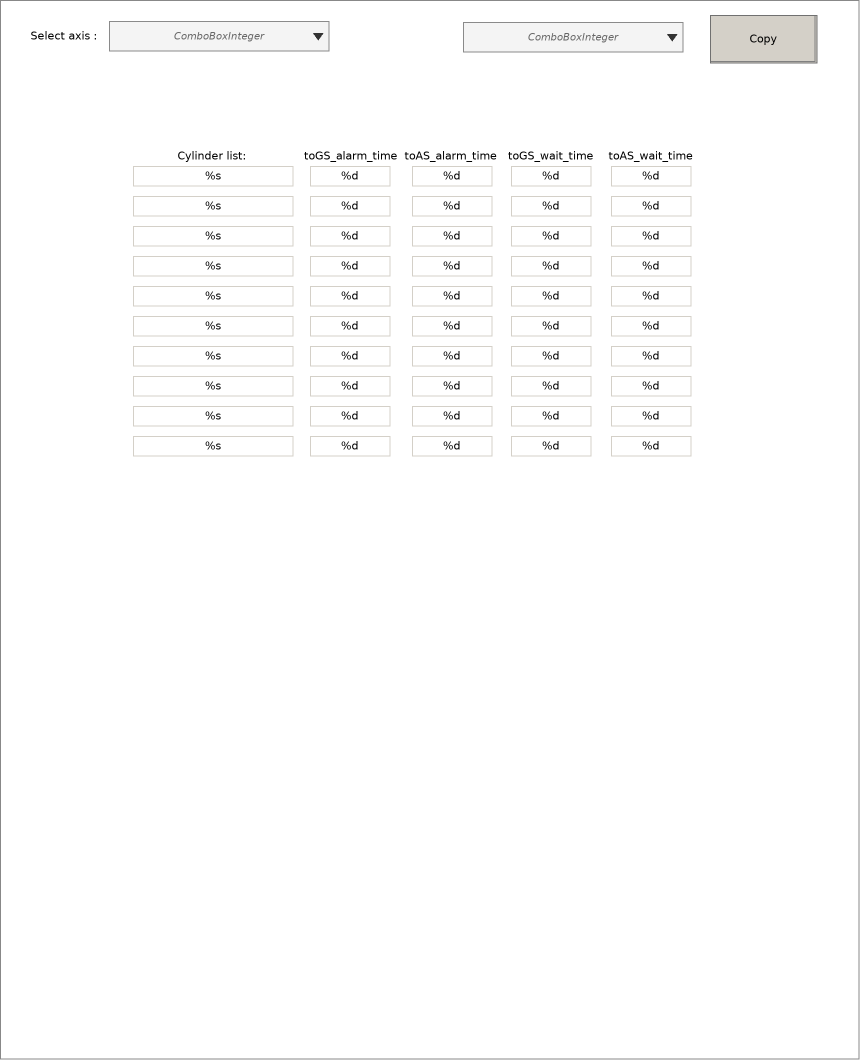
VISUALIZATION VISU_Cylinder2PosConfig  // 860x1060
    Label (165,146 94x20), "Cylinder list:"
    Label (22,21 84x30), "Select axis :"
    Label (401,146 100x20), "toAS_alarm_time"
    Label (501,146 100x20), "toGS_wait_time"
    Label (601,146 100x20), "toAS_wait_time"
    ComboBoxInteger (109,21 220x30), variable: HMI.iSelectCylinder
    Label (301,146 100x20), "toGS_alarm_time"
    Textfield (133,166 160x20), "%s", text variable: HMI.cylinderNames[HMI.iSelectCylinder][0]
    Textfield (133,196 160x20), "%s", text variable: HMI.cylinderNames[HMI.iSelectCylinder][1]
    Textfield (133,226 160x20), "%s", text variable: HMI.cylinderNames[HMI.iSelectCylinder][2]
    Textfield (133,256 160x20), "%s", text variable: HMI.cylinderNames[HMI.iSelectCylinder][3]
    Textfield (133,286 160x20), "%s", text variable: HMI.cylinderNames[HMI.iSelectCylinder][4]
    Textfield (133,316 160x20), "%s", text variable: HMI.cylinderNames[HMI.iSelectCylinder][5]
    Textfield (133,346 160x20), "%s", text variable: HMI.cylinderNames[HMI.iSelectCylinder][6]
    Textfield (133,376 160x20), "%s", text variable: HMI.cylinderNames[HMI.iSelectCylinder][7]
    Textfield (133,406 160x20), "%s", text variable: HMI.cylinderNames[HMI.iSelectCylinder][8]
    Textfield (133,436 160x20), "%s", text variable: HMI.cylinderNames[HMI.iSelectCylinder][9]
    ComboBoxInteger (463,22 220x30), variable: HMI.iSelectCylinderCopy
    Button (710,15 107x48), "Copy"
        tap HMI.btCopyCylinderCfg.button
    Textfield (310,166 80x20), "%d", text variable: _20_AUTO.recipe.cylinder2Pos[HMI.iSelectCylinder][0].toGS_alarm_time
        OnMouseDown: write the text variable via Default
    Textfield (412,166 80x20), "%d", text variable: _20_AUTO.recipe.cylinder2Pos[HMI.iSelectCylinder][0].toAS_alarm_time
        OnMouseDown: write the text variable via Default
    Textfield (511,166 80x20), "%d", text variable: _20_AUTO.recipe.cylinder2Pos[HMI.iSelectCylinder][0].toGS_wait_time
        OnMouseDown: write the text variable via Default
    Textfield (611,166 80x20), "%d", text variable: _20_AUTO.recipe.cylinder2Pos[HMI.iSelectCylinder][0].toAS_wait_time
        OnMouseDown: write the text variable via Default
    Textfield (310,196 80x20), "%d", text variable: _20_AUTO.recipe.cylinder2Pos[HMI.iSelectCylinder][1].toGS_alarm_time
        OnMouseDown: write the text variable via Default
    Textfield (412,196 80x20), "%d", text variable: _20_AUTO.recipe.cylinder2Pos[HMI.iSelectCylinder][1].toAS_alarm_time
        OnMouseDown: write the text variable via Default
    Textfield (511,196 80x20), "%d", text variable: _20_AUTO.recipe.cylinder2Pos[HMI.iSelectCylinder][1].toGS_wait_time
        OnMouseDown: write the text variable via Default
    Textfield (611,196 80x20), "%d", text variable: _20_AUTO.recipe.cylinder2Pos[HMI.iSelectCylinder][1].toAS_wait_time
        OnMouseDown: write the text variable via Default
    Textfield (310,226 80x20), "%d", text variable: _20_AUTO.recipe.cylinder2Pos[HMI.iSelectCylinder][2].toGS_alarm_time
        OnMouseDown: write the text variable via Default
    Textfield (412,226 80x20), "%d", text variable: _20_AUTO.recipe.cylinder2Pos[HMI.iSelectCylinder][2].toAS_alarm_time
        OnMouseDown: write the text variable via Default
    Textfield (511,226 80x20), "%d", text variable: _20_AUTO.recipe.cylinder2Pos[HMI.iSelectCylinder][2].toGS_wait_time
        OnMouseDown: write the text variable via Default
    Textfield (611,226 80x20), "%d", text variable: _20_AUTO.recipe.cylinder2Pos[HMI.iSelectCylinder][2].toAS_wait_time
        OnMouseDown: write the text variable via Default
    Textfield (310,256 80x20), "%d", text variable: _20_AUTO.recipe.cylinder2Pos[HMI.iSelectCylinder][3].toGS_alarm_time
        OnMouseDown: write the text variable via Default
    Textfield (412,256 80x20), "%d", text variable: _20_AUTO.recipe.cylinder2Pos[HMI.iSelectCylinder][3].toAS_alarm_time
        OnMouseDown: write the text variable via Default
    Textfield (511,256 80x20), "%d", text variable: _20_AUTO.recipe.cylinder2Pos[HMI.iSelectCylinder][3].toGS_wait_time
        OnMouseDown: write the text variable via Default
    Textfield (611,256 80x20), "%d", text variable: _20_AUTO.recipe.cylinder2Pos[HMI.iSelectCylinder][3].toAS_wait_time
        OnMouseDown: write the text variable via Default
    Textfield (310,286 80x20), "%d", text variable: _20_AUTO.recipe.cylinder2Pos[HMI.iSelectCylinder][4].toGS_alarm_time
        OnMouseDown: write the text variable via Default
    Textfield (412,286 80x20), "%d", text variable: _20_AUTO.recipe.cylinder2Pos[HMI.iSelectCylinder][4].toAS_alarm_time
        OnMouseDown: write the text variable via Default
    Textfield (511,286 80x20), "%d", text variable: _20_AUTO.recipe.cylinder2Pos[HMI.iSelectCylinder][4].toGS_wait_time
        OnMouseDown: write the text variable via Default
    Textfield (611,286 80x20), "%d", text variable: _20_AUTO.recipe.cylinder2Pos[HMI.iSelectCylinder][4].toAS_wait_time
        OnMouseDown: write the text variable via Default
    Textfield (310,316 80x20), "%d", text variable: _20_AUTO.recipe.cylinder2Pos[HMI.iSelectCylinder][5].toGS_alarm_time
        OnMouseDown: write the text variable via Default
    Textfield (412,316 80x20), "%d", text variable: _20_AUTO.recipe.cylinder2Pos[HMI.iSelectCylinder][5].toAS_alarm_time
        OnMouseDown: write the text variable via Default
    Textfield (511,316 80x20), "%d", text variable: _20_AUTO.recipe.cylinder2Pos[HMI.iSelectCylinder][5].toGS_wait_time
        OnMouseDown: write the text variable via Default
    Textfield (611,316 80x20), "%d", text variable: _20_AUTO.recipe.cylinder2Pos[HMI.iSelectCylinder][5].toAS_wait_time
        OnMouseDown: write the text variable via Default
    Textfield (310,346 80x20), "%d", text variable: _20_AUTO.recipe.cylinder2Pos[HMI.iSelectCylinder][6].toGS_alarm_time
        OnMouseDown: write the text variable via Default
    Textfield (412,346 80x20), "%d", text variable: _20_AUTO.recipe.cylinder2Pos[HMI.iSelectCylinder][6].toAS_alarm_time
        OnMouseDown: write the text variable via Default
    Textfield (511,346 80x20), "%d", text variable: _20_AUTO.recipe.cylinder2Pos[HMI.iSelectCylinder][6].toGS_wait_time
        OnMouseDown: write the text variable via Default
    Textfield (611,346 80x20), "%d", text variable: _20_AUTO.recipe.cylinder2Pos[HMI.iSelectCylinder][6].toAS_wait_time
        OnMouseDown: write the text variable via Default
    Textfield (310,376 80x20), "%d", text variable: _20_AUTO.recipe.cylinder2Pos[HMI.iSelectCylinder][7].toGS_alarm_time
        OnMouseDown: write the text variable via Default
    Textfield (412,376 80x20), "%d", text variable: _20_AUTO.recipe.cylinder2Pos[HMI.iSelectCylinder][7].toAS_alarm_time
        OnMouseDown: write the text variable via Default
    Textfield (511,376 80x20), "%d", text variable: _20_AUTO.recipe.cylinder2Pos[HMI.iSelectCylinder][7].toGS_wait_time
        OnMouseDown: write the text variable via Default
    Textfield (611,376 80x20), "%d", text variable: _20_AUTO.recipe.cylinder2Pos[HMI.iSelectCylinder][7].toAS_wait_time
        OnMouseDown: write the text variable via Default
    Textfield (310,406 80x20), "%d", text variable: _20_AUTO.recipe.cylinder2Pos[HMI.iSelectCylinder][8].toGS_alarm_time
        OnMouseDown: write the text variable via Default
    Textfield (412,406 80x20), "%d", text variable: _20_AUTO.recipe.cylinder2Pos[HMI.iSelectCylinder][8].toAS_alarm_time
        OnMouseDown: write the text variable via Default
    Textfield (511,406 80x20), "%d", text variable: _20_AUTO.recipe.cylinder2Pos[HMI.iSelectCylinder][8].toGS_wait_time
        OnMouseDown: write the text variable via Default
    Textfield (611,406 80x20), "%d", text variable: _20_AUTO.recipe.cylinder2Pos[HMI.iSelectCylinder][8].toAS_wait_time
        OnMouseDown: write the text variable via Default
    Textfield (310,436 80x20), "%d", text variable: _20_AUTO.recipe.cylinder2Pos[HMI.iSelectCylinder][9].toGS_alarm_time
        OnMouseDown: write the text variable via Default
    Textfield (412,436 80x20), "%d", text variable: _20_AUTO.recipe.cylinder2Pos[HMI.iSelectCylinder][9].toAS_alarm_time
        OnMouseDown: write the text variable via Default
    Textfield (511,436 80x20), "%d", text variable: _20_AUTO.recipe.cylinder2Pos[HMI.iSelectCylinder][9].toGS_wait_time
        OnMouseDown: write the text variable via Default
    Textfield (611,436 80x20), "%d", text variable: _20_AUTO.recipe.cylinder2Pos[HMI.iSelectCylinder][9].toAS_wait_time
        OnMouseDown: write the text variable via Default
END_VISUALIZATION

(* stored: Version 1.1.0.1, ProductVersion 3.1.4024.6
   Visu VISU_Cylinder2PosConfig: Id {a8963da2-2a50-4181-88cd-94b3efd1f47f} *)
